// Mitsubishi GX Works2 project: plc_new   PLC: FX3G

// global labels: Global1
VAR_GLOBAL
  startDay AT X007 : BOOL;
END_VAR
VAR_GLOBAL CONSTANT
  const0 : INT;
END_VAR
VAR_GLOBAL
  analog_output AT D8282 : INT;
  total_gummyGam_packages AT D1170 : REAL;
END_VAR
VAR_GLOBAL CONSTANT
  constant_0 : REAL;
END_VAR
VAR_GLOBAL
  input_rasp AT D7000 : REAL;
  raspberry_inventory AT D1130 : REAL;
  input_lemon AT D7010 : REAL;
  lemon_inventory AT D1140 : REAL;
  input_stabilizer AT D7020 : REAL;
  stabilizer_inventory AT D1150 : REAL;
  gummybears_inventory AT D1160 : REAL;
  input_gummybear AT D7030 : REAL;
  not_the_1st_iter AT M23 : BOOL;
END_VAR
VAR_GLOBAL CONSTANT
  regular_raspberry_req : REAL := 280;
END_VAR
VAR_GLOBAL
  enough_raspberry_regular AT M20 : BOOL;
END_VAR
VAR_GLOBAL CONSTANT
  regular_lemon_req : REAL := 455;
END_VAR
VAR_GLOBAL
  enough_lemon_regular AT M21 : BOOL;
END_VAR
VAR_GLOBAL CONSTANT
  regular_stabilizer_req : REAL := 105;
END_VAR
VAR_GLOBAL
  enough_stabilizer_regular AT M22 : BOOL;
END_VAR
VAR_GLOBAL CONSTANT
  regular_gummybears_req : REAL := 28;
END_VAR
VAR_GLOBAL
  enough_gummybears_regular AT M24 : BOOL;
  possible_making_regular AT M4 : BOOL;
END_VAR
VAR_GLOBAL CONSTANT
  pinuk_raspberry_req : REAL := 385;
END_VAR
VAR_GLOBAL
  enough_raspberry_pinuk AT M30 : BOOL;
END_VAR
VAR_GLOBAL CONSTANT
  pinuk_lemon_req : REAL := 665;
END_VAR
VAR_GLOBAL
  enough_lemon_pinuk AT M31 : BOOL;
END_VAR
VAR_GLOBAL CONSTANT
  pinuk_stabilizer_req : REAL := 210;
END_VAR
VAR_GLOBAL
  enough_stabilizer_pinuk AT M32 : BOOL;
END_VAR
VAR_GLOBAL CONSTANT
  pinuk_gummybears_req : REAL := 70;
END_VAR
VAR_GLOBAL
  enough_gummybears_pinuk AT M33 : BOOL;
  possible_making_pinuk AT M5 : BOOL;
  endDay AT X005 : BOOL;
  ongoingDay AT Y007 : BOOL;
  analog_input AT D8280 : INT;
  analog_input_res AT D1700 : REAL;
END_VAR
VAR_GLOBAL CONSTANT
  const_400 : REAL := 400;
END_VAR
VAR_GLOBAL
  start_packing_cone AT X004 : BOOL;
  pack_a_cone AT X000 : BOOL;
END_VAR
VAR_GLOBAL CONSTANT
  constant5 : REAL := 5;
  constant6 : REAL := 6;
END_VAR
VAR_GLOBAL
  regular AT M2 : BOOL;
  pinuk AT M3 : BOOL;
END_VAR
VAR_GLOBAL CONSTANT
  constant_350 : REAL := 350;
END_VAR
VAR_GLOBAL
  raspberry_iceCream_container AT D2000 : REAL;
  lemon_iceCream_container AT D2010 : REAL;
END_VAR
VAR_GLOBAL CONSTANT
  constant_560 : REAL := 560;
  constant_700 : REAL := 700;
END_VAR
VAR_GLOBAL
  making_iceCream_inProcess AT Y000 : BOOL;
  finish_making_iceCream_timer AT TS1 : BOOL;
  process_timer AT TC1 : BOOL;
END_VAR
VAR_GLOBAL CONSTANT
  constant_50 : INT := 50;
END_VAR
VAR_GLOBAL
  start_freezing AT X002 : BOOL;
  freezing_in_process AT Y002 : BOOL;
END_VAR
VAR_GLOBAL CONSTANT
  freezing_time_8sec : INT := 80;
END_VAR
VAR_GLOBAL
  temp_sensor AT X003 : BOOL;
  start_regular_mixing_timer AT TC4 : BOOL;
END_VAR
VAR_GLOBAL CONSTANT
  regular_mixing_time_3sec : WORD := 30;
END_VAR
VAR_GLOBAL
  startpinuk_miking_timer AT TC5 : BOOL;
END_VAR
VAR_GLOBAL CONSTANT
  pinuk_mixing_time_5sec : WORD := 50;
  constant_868 : REAL := 868;
  constant_1330 : REAL := 1330;
END_VAR
VAR_GLOBAL
  end_regular_mixing_timer AT TS4 : BOOL;
  end_pinuk_mixing_timer AT TS5 : BOOL;
  end_mixing_help_bulb AT M6 : BOOL;
  blink_round AT M8 : BOOL;
  bulb6_on AT TC6 : BOOL;
END_VAR
VAR_GLOBAL CONSTANT
  blink_time : INT := 5;
END_VAR
VAR_GLOBAL
  bulb6_off AT TS6 : BOOL;
  bulb_y6 AT Y006 : BOOL;
  bulb5_on AT TC7 : BOOL;
  bulb5_off AT TS7 : BOOL;
  bulb_y5 AT Y005 : BOOL;
  cooling_finish AT M36 : BOOL;
  start_freezing_timer AT TC3 : BOOL;
  finish_freezing_timer AT TS3 : BOOL;
  cooling_finish_by_temp AT M35 : BOOL;
  regular_in_process AT M40 : BOOL;
  pinuk_in_process AT M41 : BOOL;
  mixing_container AT D2040 : REAL;
  start_making_flavors AT X001 : BOOL;
  raspberry_freezing_container AT D2020 : REAL;
  lemon_freezing_container AT D2030 : REAL;
  finish_count_cones AT CS1 : BOOL;
  count_7cones_in_pack AT CC1 : BOOL;
END_VAR
VAR_GLOBAL CONSTANT
  constant_7 : INT := 7;
END_VAR
VAR_GLOBAL
  packing_bulb AT Y004 : BOOL;
END_VAR
VAR_GLOBAL CONSTANT
  constant_1 : REAL := 1;
  constant_div_7 : REAL := 7;
END_VAR
VAR_GLOBAL
  div_material_per_con AT D2050 : REAL;
END_VAR
VAR_GLOBAL CONSTANT
  constant_490 : REAL := 490;
END_VAR
VAR_GLOBAL
  end_packing AT M50 : BOOL;
END_VAR
VAR_GLOBAL CONSTANT
  constant_40 : REAL := 40;
END_VAR
VAR_GLOBAL
  total_packages AT D2060 : REAL;
END_VAR

// task Task_01 (event TRUE, interval 0, priority 31): POU_01

PROGRAM POU_01
(* structured ladder/FBD written out as ST: instructions are called as NAME(EN, inputs, outputs); _pN, _eN, _tN stand for wires *)
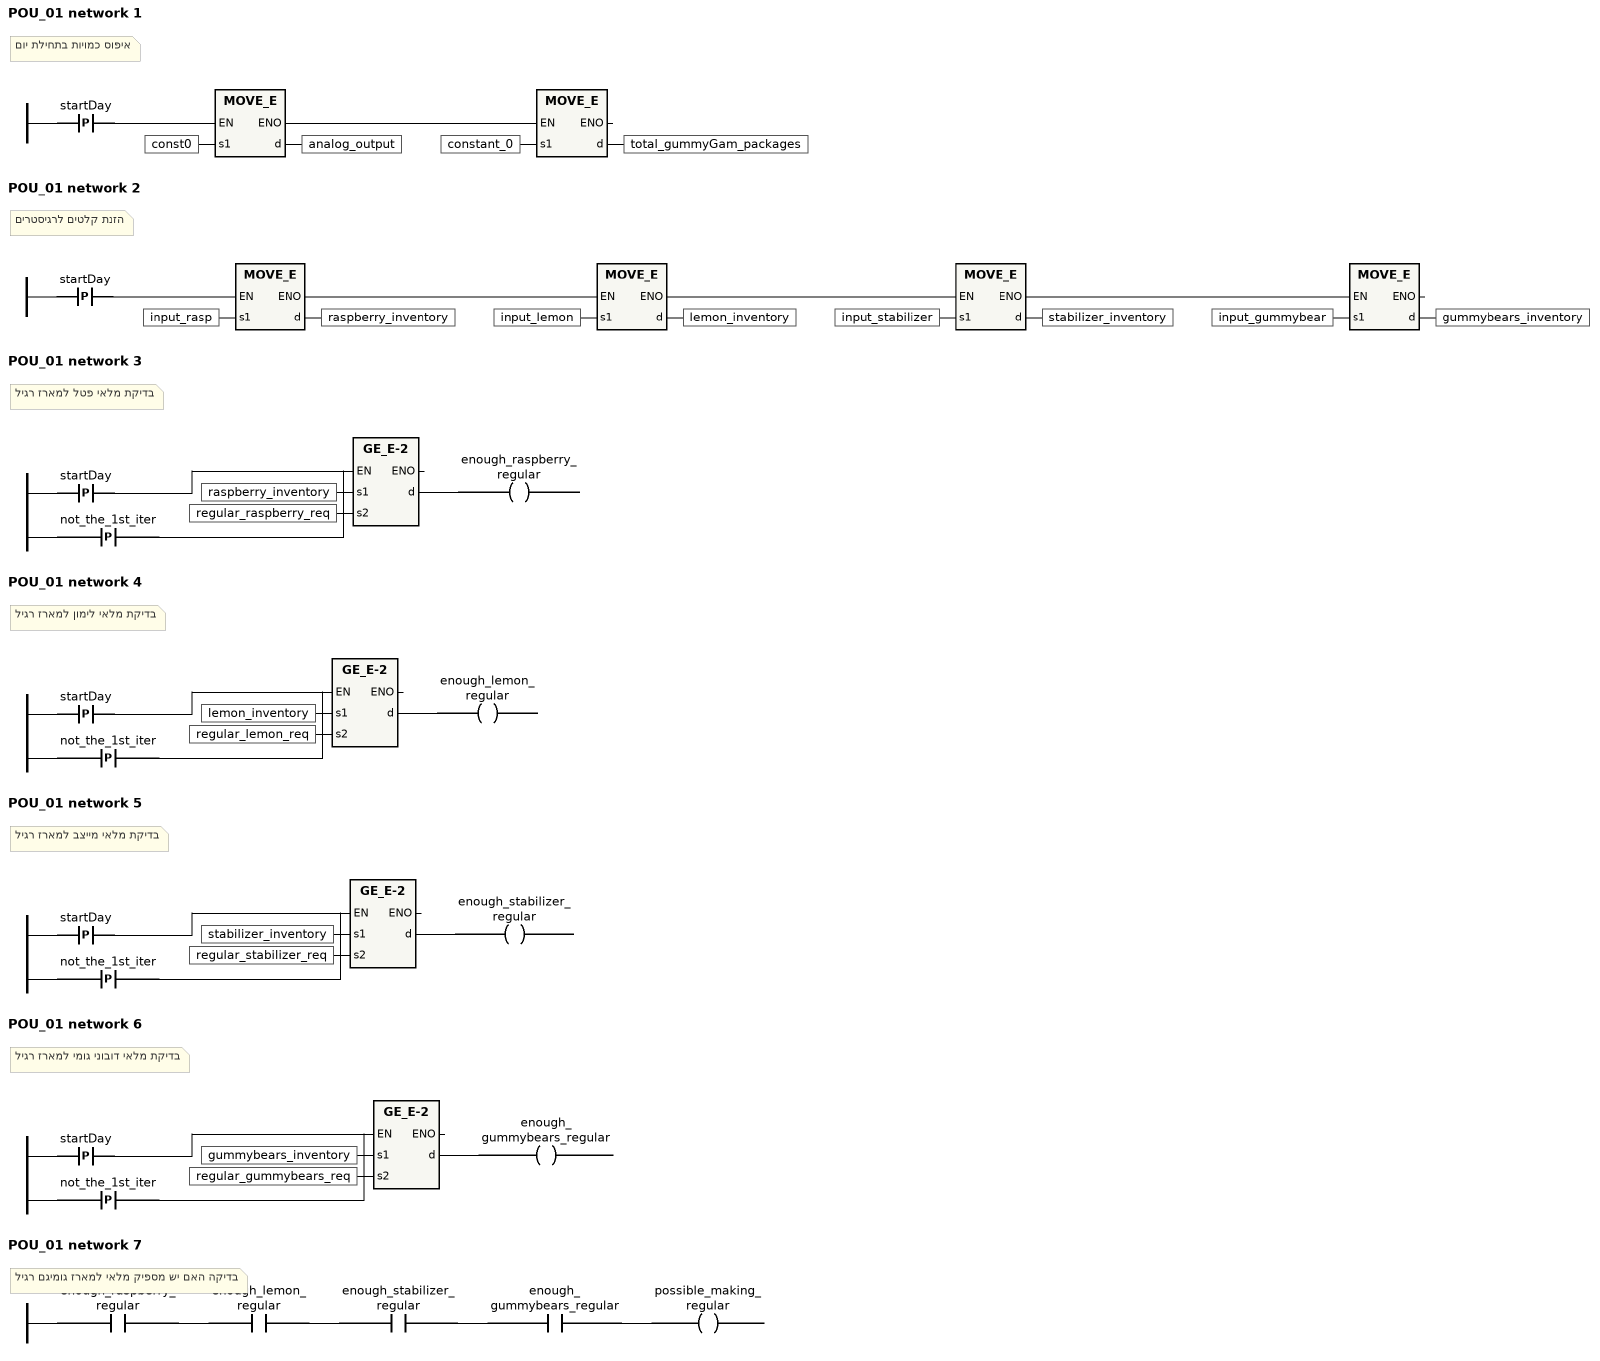
(* network 1 *)
(* איפוס כמויות בתחילת יום *)
_e1 := MOVE_E(LDP(TRUE, startDay), const0, analog_output);
MOVE_E(_e1, constant_0, total_gummyGam_packages);
(* network 2 *)
(* הזנת קלטים לרגיסטרים *)
_e1 := MOVE_E(LDP(TRUE, startDay), input_rasp, raspberry_inventory);
_e2 := MOVE_E(_e1, input_lemon, lemon_inventory);
_e3 := MOVE_E(_e2, input_stabilizer, stabilizer_inventory);
MOVE_E(_e3, input_gummybear, gummybears_inventory);
(* network 3 *)
(* בדיקת מלאי פטל למארז רגיל *)
GE_E(LDP(TRUE, startDay) OR LDP(TRUE, not_the_1st_iter), raspberry_inventory, regular_raspberry_req, _t1);
enough_raspberry_regular := _t1;
(* network 4 *)
(* בדיקת מלאי לימון למארז רגיל *)
GE_E(LDP(TRUE, startDay) OR LDP(TRUE, not_the_1st_iter), lemon_inventory, regular_lemon_req, _t1);
enough_lemon_regular := _t1;
(* network 5 *)
(* בדיקת מלאי מייצב למארז רגיל *)
GE_E(LDP(TRUE, startDay) OR LDP(TRUE, not_the_1st_iter), stabilizer_inventory, regular_stabilizer_req, _t1);
enough_stabilizer_regular := _t1;
(* network 6 *)
(* בדיקת מלאי דובוני גומי למארז רגיל *)
GE_E(LDP(TRUE, startDay) OR LDP(TRUE, not_the_1st_iter), gummybears_inventory, regular_gummybears_req, _t1);
enough_gummybears_regular := _t1;
(* network 7 *)
(* בדיקה האם יש מספיק מלאי למארז גומיגם רגיל *)
possible_making_regular := enough_raspberry_regular AND enough_lemon_regular AND enough_stabilizer_regular AND enough_gummybears_regular;
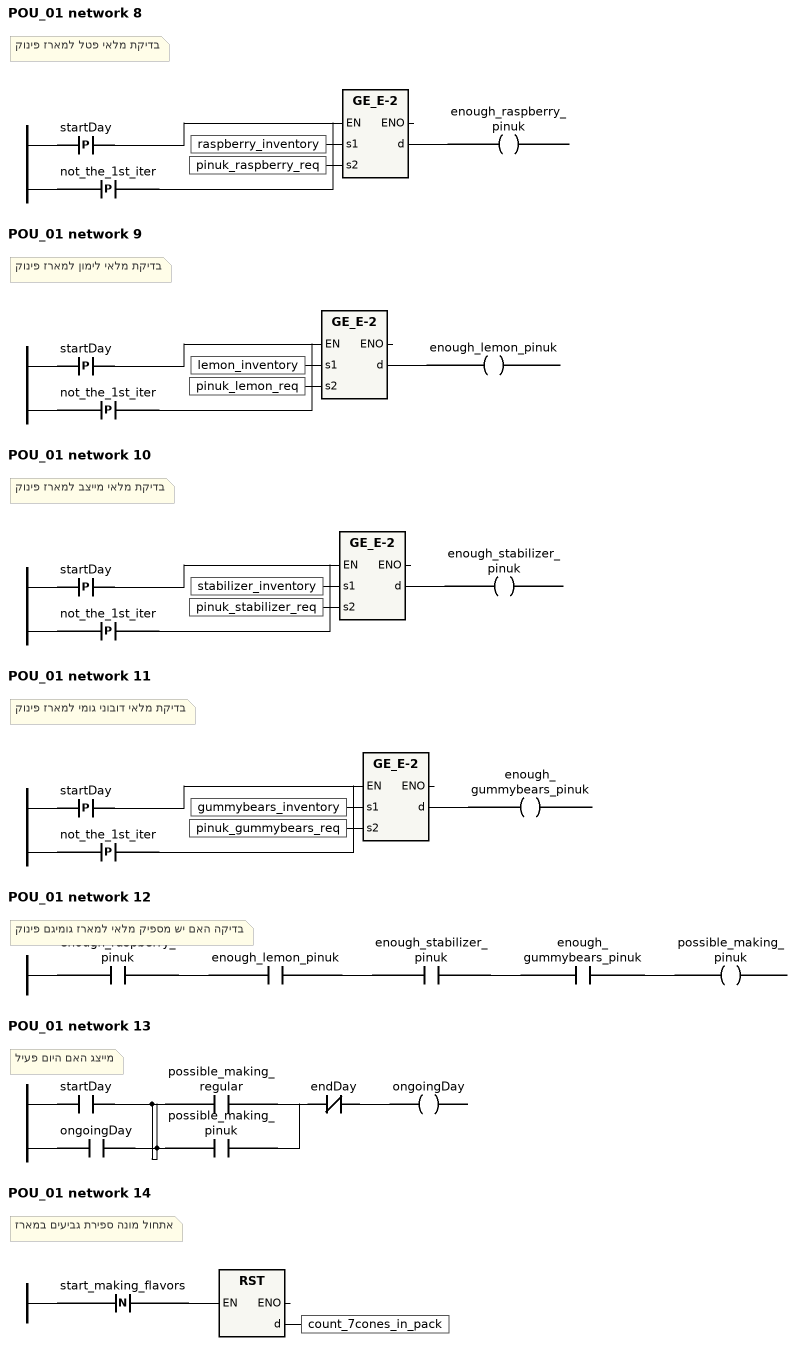
(* network 8 *)
(* בדיקת מלאי פטל למארז פינוק *)
GE_E(LDP(TRUE, startDay) OR LDP(TRUE, not_the_1st_iter), raspberry_inventory, pinuk_raspberry_req, _t1);
enough_raspberry_pinuk := _t1;
(* network 9 *)
(* בדיקת מלאי לימון למארז פינוק *)
GE_E(LDP(TRUE, startDay) OR LDP(TRUE, not_the_1st_iter), lemon_inventory, pinuk_lemon_req, _t1);
enough_lemon_pinuk := _t1;
(* network 10 *)
(* בדיקת מלאי מייצב למארז פינוק *)
GE_E(LDP(TRUE, startDay) OR LDP(TRUE, not_the_1st_iter), stabilizer_inventory, pinuk_stabilizer_req, _t1);
enough_stabilizer_pinuk := _t1;
(* network 11 *)
(* בדיקת מלאי דובוני גומי למארז פינוק *)
GE_E(LDP(TRUE, startDay) OR LDP(TRUE, not_the_1st_iter), gummybears_inventory, pinuk_gummybears_req, _t1);
enough_gummybears_pinuk := _t1;
(* network 12 *)
(* בדיקה האם יש מספיק מלאי למארז גומיגם פינוק *)
possible_making_pinuk := enough_raspberry_pinuk AND enough_lemon_pinuk AND enough_stabilizer_pinuk AND enough_gummybears_pinuk;
(* network 13 *)
(* מייצג האם היום פעיל *)
_p1 := startDay OR ongoingDay;
ongoingDay := ((_p1 AND possible_making_regular) OR (_p1 AND possible_making_pinuk)) AND NOT endDay;
(* network 14 *)
(* אתחול מונה ספירת גביעים במארז *)
RST(LDF(TRUE, start_making_flavors), count_7cones_in_pack);
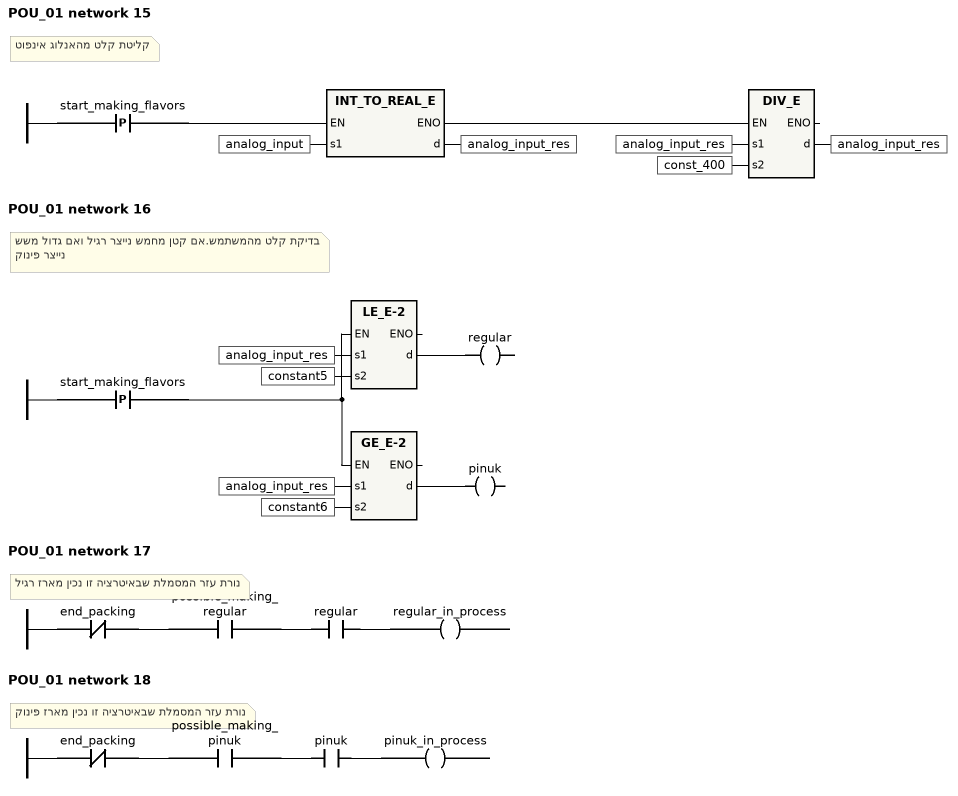
(* network 15 *)
(* קליטת קלט מהאנלוג אינפוט *)
_e1 := INT_TO_REAL_E(LDP(TRUE, start_making_flavors), analog_input, analog_input_res);
DIV_E(_e1, analog_input_res, const_400, analog_input_res);
(* network 16 *)
(* בדיקת קלט מהמשתמש.אם קטן מחמש נייצר רגיל ואם גדול משש נייצר פינוק *)
_p1 := LDP(TRUE, start_making_flavors);
LE_E(_p1, analog_input_res, constant5, _t2);
regular := _t2;
GE_E(_p1, analog_input_res, constant6, _t3);
pinuk := _t3;
(* network 17 *)
(* נורת עזר המסמלת שבאיטרציה זו נכין מארז רגיל *)
regular_in_process := NOT end_packing AND possible_making_regular AND regular;
(* network 18 *)
(* נורת עזר המסמלת שבאיטרציה זו נכין מארז פינוק *)
pinuk_in_process := NOT end_packing AND possible_making_pinuk AND pinuk;
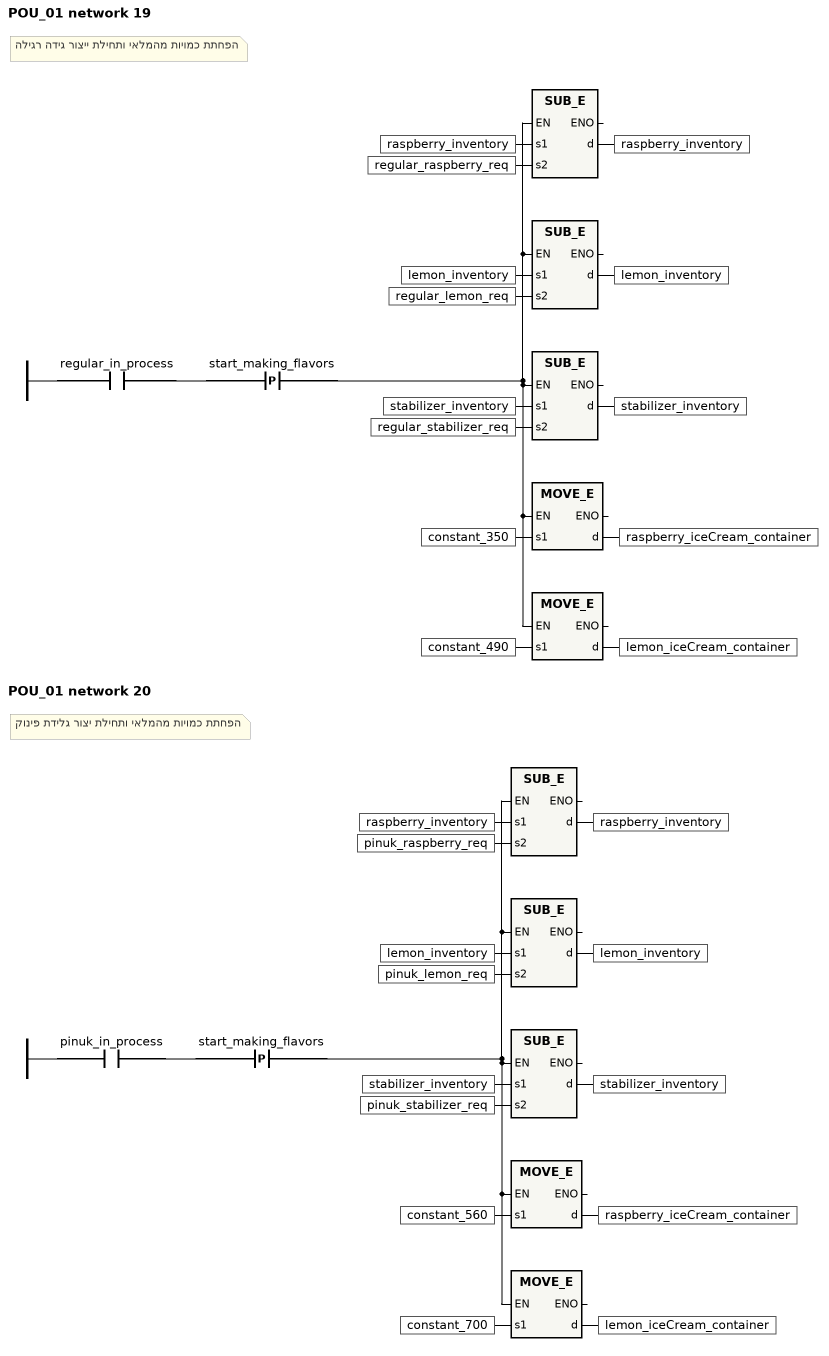
(* network 19 *)
(* הפחתת כמויות מהמלאי ותחילת ייצור גידה רגילה *)
_p1 := regular_in_process AND LDP(TRUE, start_making_flavors);
SUB_E(_p1, raspberry_inventory, regular_raspberry_req, raspberry_inventory);
SUB_E(_p1, lemon_inventory, regular_lemon_req, lemon_inventory);
SUB_E(_p1, stabilizer_inventory, regular_stabilizer_req, stabilizer_inventory);
MOVE_E(_p1, constant_350, raspberry_iceCream_container);
MOVE_E(_p1, constant_490, lemon_iceCream_container);
(* network 20 *)
(* הפחתת כמויות מהמלאי ותחילת יצור גלידת פינוק *)
_p1 := pinuk_in_process AND LDP(TRUE, start_making_flavors);
SUB_E(_p1, raspberry_inventory, pinuk_raspberry_req, raspberry_inventory);
SUB_E(_p1, lemon_inventory, pinuk_lemon_req, lemon_inventory);
SUB_E(_p1, stabilizer_inventory, pinuk_stabilizer_req, stabilizer_inventory);
MOVE_E(_p1, constant_560, raspberry_iceCream_container);
MOVE_E(_p1, constant_700, lemon_iceCream_container);
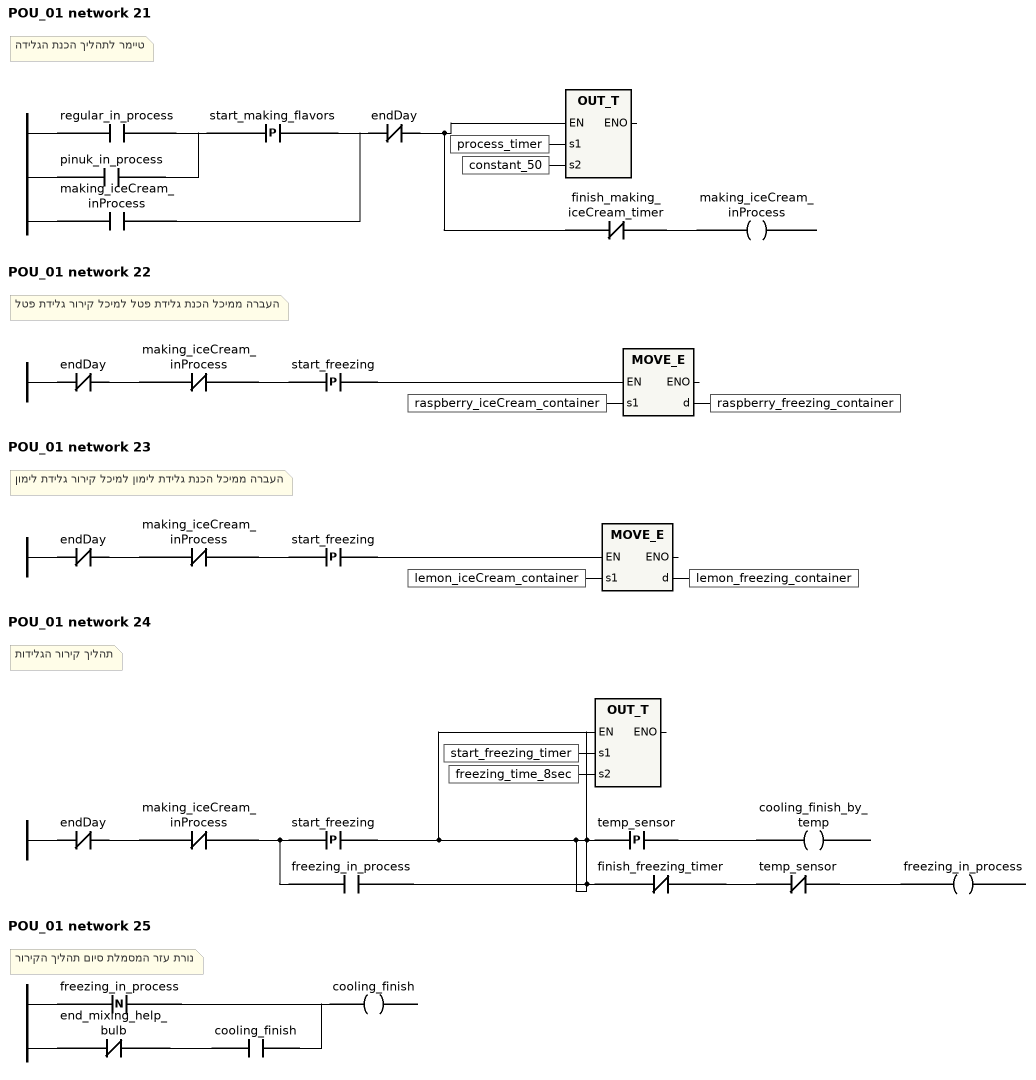
(* network 21 *)
(* טיימר לתהליך הכנת הגלידה *)
_p1 := (((regular_in_process OR pinuk_in_process) AND LDP(TRUE, start_making_flavors)) OR making_iceCream_inProcess) AND NOT endDay;
making_iceCream_inProcess := _p1 AND NOT finish_making_iceCream_timer;
OUT_T(_p1, process_timer, constant_50);
(* network 22 *)
(* העברה ממיכל הכנת גלידת פטל למיכל קירור גלידת פטל *)
MOVE_E(NOT endDay AND NOT making_iceCream_inProcess AND LDP(TRUE, start_freezing), raspberry_iceCream_container, raspberry_freezing_container);
(* network 23 *)
(* העברה ממיכל הכנת גלידת לימון למיכל קירור גלידת לימון *)
MOVE_E(NOT endDay AND NOT making_iceCream_inProcess AND LDP(TRUE, start_freezing), lemon_iceCream_container, lemon_freezing_container);
(* network 24 *)
(* תהליך קירור הגלידות *)
_p1 := NOT endDay AND NOT making_iceCream_inProcess;
_p2 := (_p1 AND LDP(TRUE, start_freezing)) OR (_p1 AND freezing_in_process);
OUT_T(_p2, start_freezing_timer, freezing_time_8sec);
cooling_finish_by_temp := _p2 AND LDP(TRUE, temp_sensor);
freezing_in_process := _p2 AND NOT finish_freezing_timer AND NOT temp_sensor;
(* network 25 *)
(* נורת עזר המסמלת סיום תהליך הקירור *)
cooling_finish := LDF(TRUE, freezing_in_process) OR (NOT end_mixing_help_bulb AND cooling_finish);
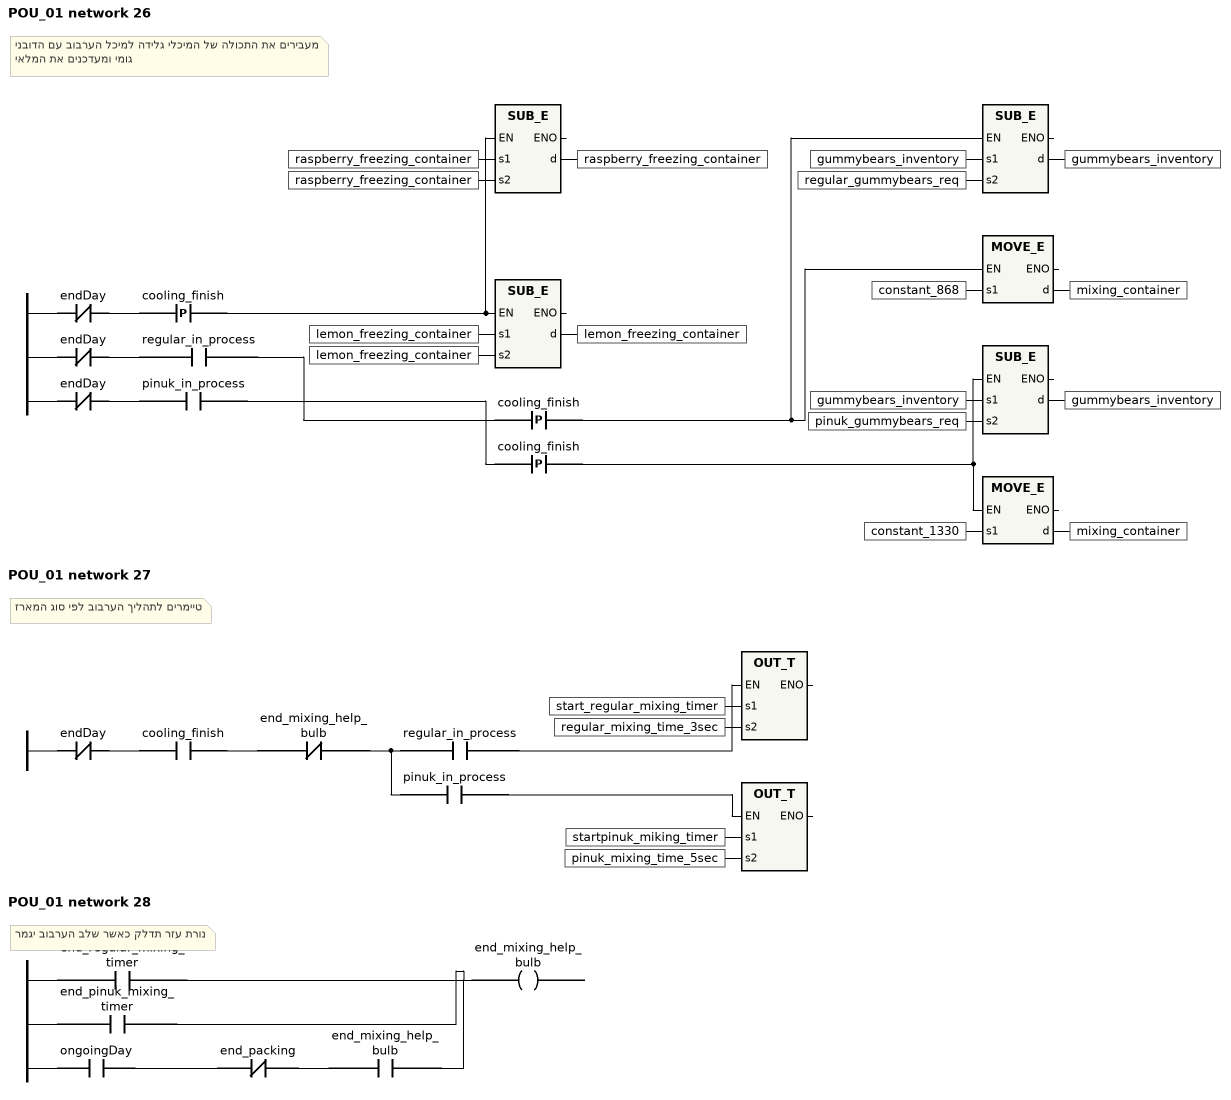
(* network 26 *)
(* מעבירים את התכולה של המיכלי גלידה למיכל הערבוב עם הדובני גומי ומעדכנים את המלאי *)
_p1 := NOT endDay AND LDP(TRUE, cooling_finish);
SUB_E(_p1, raspberry_freezing_container, raspberry_freezing_container, raspberry_freezing_container);
SUB_E(_p1, lemon_freezing_container, lemon_freezing_container, lemon_freezing_container);
_p2 := NOT endDay AND regular_in_process AND LDP(TRUE, cooling_finish);
SUB_E(_p2, gummybears_inventory, regular_gummybears_req, gummybears_inventory);
MOVE_E(_p2, constant_868, mixing_container);
_p3 := NOT endDay AND pinuk_in_process AND LDP(TRUE, cooling_finish);
SUB_E(_p3, gummybears_inventory, pinuk_gummybears_req, gummybears_inventory);
MOVE_E(_p3, constant_1330, mixing_container);
(* network 27 *)
(* טיימרים לתהליך הערבוב לפי סוג המארז *)
_p1 := NOT endDay AND cooling_finish AND NOT end_mixing_help_bulb;
OUT_T(_p1 AND regular_in_process, start_regular_mixing_timer, regular_mixing_time_3sec);
OUT_T(_p1 AND pinuk_in_process, startpinuk_miking_timer, pinuk_mixing_time_5sec);
(* network 28 *)
(* נורת עזר תדלק כאשר שלב הערבוב יגמר *)
end_mixing_help_bulb := end_regular_mixing_timer OR end_pinuk_mixing_timer OR (ongoingDay AND NOT end_packing AND end_mixing_help_bulb);
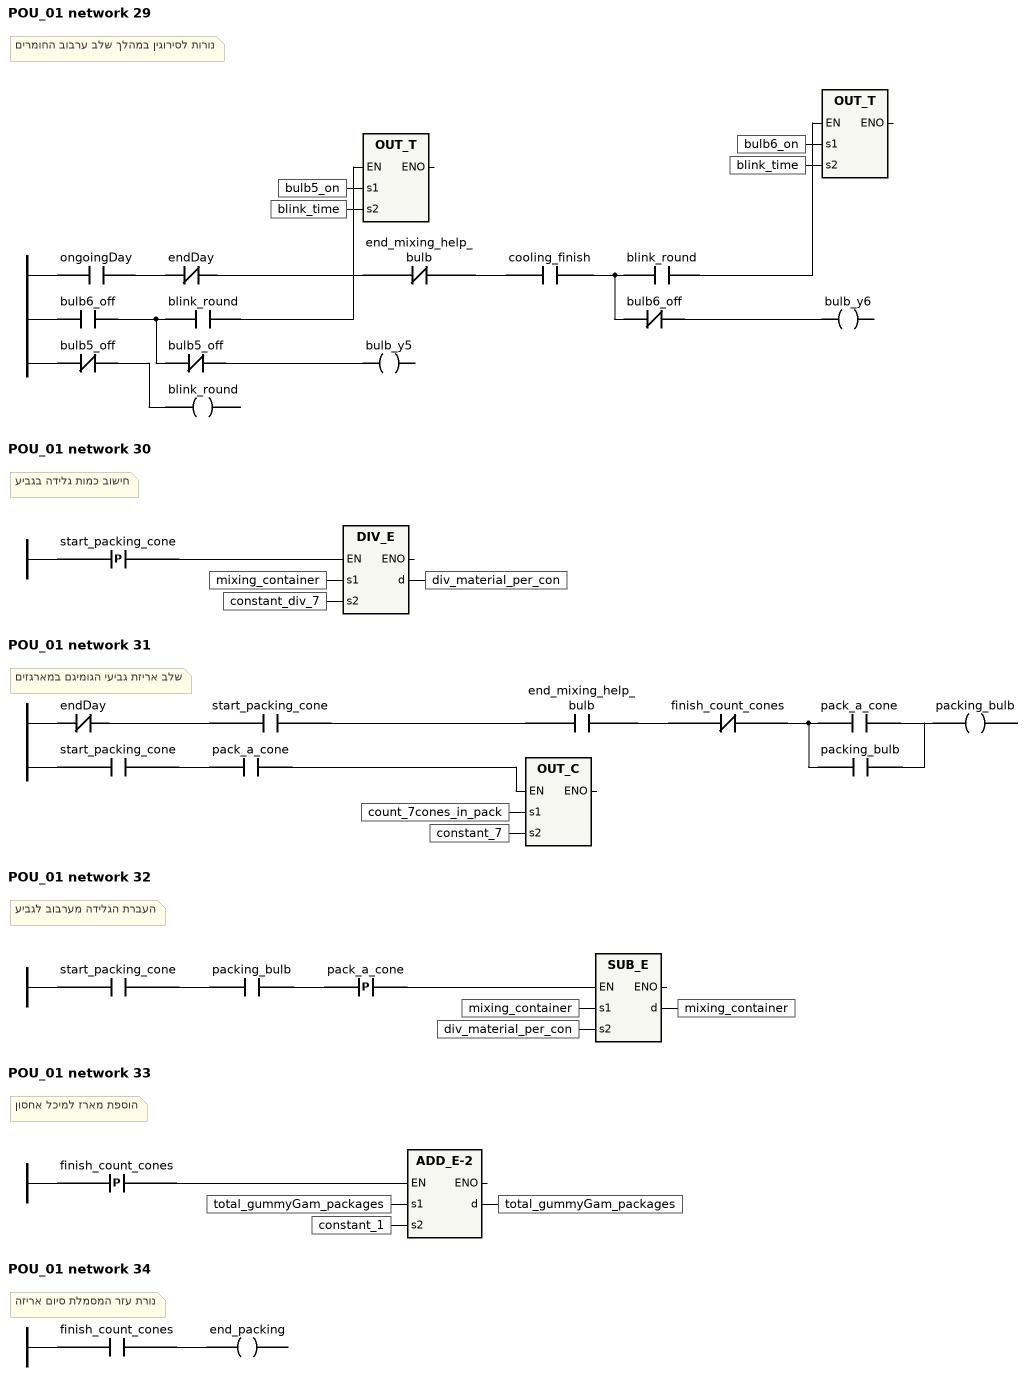
(* network 29 *)
(* נורות לסירוגין במהלך שלב ערבוב החומרים *)
_p1 := ongoingDay AND NOT endDay AND NOT end_mixing_help_bulb AND cooling_finish;
OUT_T(_p1 AND blink_round, bulb6_on, blink_time);
bulb_y6 := _p1 AND NOT bulb6_off;
OUT_T(bulb6_off AND blink_round, bulb5_on, blink_time);
bulb_y5 := bulb6_off AND NOT bulb5_off;
blink_round := NOT bulb5_off;
(* network 30 *)
(* חישוב כמות גלידה בגביע *)
DIV_E(LDP(TRUE, start_packing_cone), mixing_container, constant_div_7, div_material_per_con);
(* network 31 *)
(* שלב אריזת גביעי הגומיגם במארגזים *)
_p1 := NOT endDay AND start_packing_cone AND end_mixing_help_bulb AND NOT finish_count_cones;
packing_bulb := (_p1 AND pack_a_cone) OR (_p1 AND packing_bulb);
OUT_C(start_packing_cone AND pack_a_cone, count_7cones_in_pack, constant_7);
(* network 32 *)
(* העברת הגלידה מערבוב לגביע *)
SUB_E(start_packing_cone AND packing_bulb AND LDP(TRUE, pack_a_cone), mixing_container, div_material_per_con, mixing_container);
(* network 33 *)
(* הוספת מארז למיכל אחסון *)
ADD_E(LDP(TRUE, finish_count_cones), total_gummyGam_packages, constant_1, total_gummyGam_packages);
(* network 34 *)
(* נורת עזר המסמלת סיום אריזה *)
end_packing := finish_count_cones;
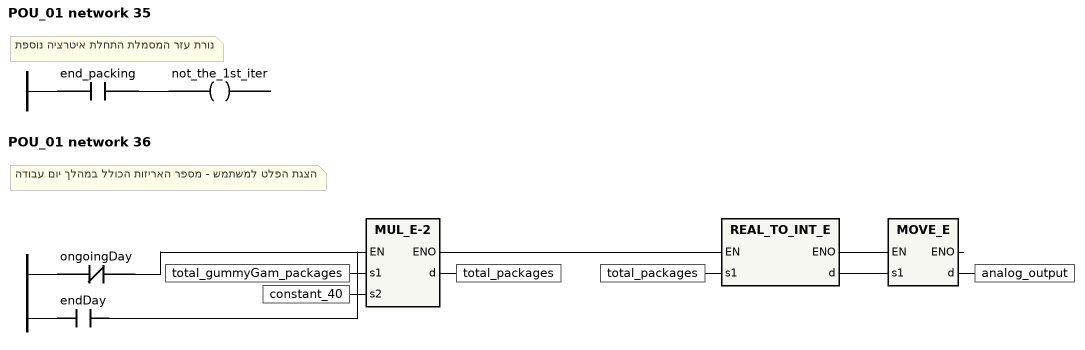
(* network 35 *)
(* נורת עזר המסמלת התחלת איטרציה נוספת *)
not_the_1st_iter := end_packing;
(* network 36 *)
(* הצגת הפלט למשתמש - מספר האריזות הכולל במהלך יום עבודה *)
_e1 := MUL_E((NOT ongoingDay) OR endDay, total_gummyGam_packages, constant_40, total_packages);
_e3 := REAL_TO_INT_E(_e1, total_packages, _t2);
MOVE_E(_e3, _t2, analog_output);
END_PROGRAM
